TYPE ST_TopMoldErrors_OLD :
STRUCT
	Hydraulic					: ST_HydraulicErrorsAnalog;
	HeatingZone 				: ARRAY [1..6] OF ST_HeatingZoneErrors;
END_STRUCT
END_TYPE

(* stored: Version 1.1.0.1, ProductVersion 3.1.4020.12
   DUT ST_TopMoldErrors_OLD: Id {f2615682-490c-4c89-af9c-9e4e15590e22} *)
